(* IEC 61131-3 sources: PLC_structured_text/, 3 files *)

(* ---- electrical_motor.st ---- *)
PROGRAM Main
VAR
	AI_FRQ	AT %IW2: INT;
	AO_FRQ	AT %QW2: INT;
	DI_RUN	AT %IX0.0: BOOL;
	DI_ERR	AT %IX0.1: BOOL;
	DI_AUTO	AT %IX0.2: BOOL;
	DO_RUN	AT %QX0.0: BOOL;
	DO_FWD	AT %QX0.4: BOOL;
	DO_BKW	AT %QX0.5: BOOL;
	EN_AI_HZ	AT %QX1.1: BOOL;
	Control_Mode	AT %MW0: INT;
	HMI_SHOW_Hz	AT %MW1: INT;
	HMI_SHOW_Err	AT %MW2: INT;
	HMI_SHOW_RUN	AT %MW3: INT;
	HMI_SHOW_NONE	AT %MW4: INT;
	HMI_SET_FWD	AT %MW6: INT;
	HMI_SET_BCK	AT %MW7: INT;
	HMI_SET_Fr_GiveAQ AT %MW10: INT;
	RUN_TIME AT %MD11: REAL;
	HMI_SET_FR	AT %MD12: REAL;
	CurveSet_Hz	: REAL;
	CurveSet_Count : DINT;
	BLINK01 : BLINK;
	BLINK02 : BLINK;
	BLINK03 : BLINK;
	R_TRIG01 : R_TRIG;
	R_TRIG02 : R_TRIG;
	R_TRIG03 : R_TRIG;

	Run_count: DINT;
	Run_fre: REAL;
END_VAR

HMI_SHOW_Hz	:= AI_FRQ;
IF HMI_SET_FR >= 0.0 AND HMI_SET_FR <= 50.0 THEN
	HMI_SET_Fr_GiveAQ := REAL_TO_INT(HMI_SET_FR * 100.0);
END_IF
CASE control_mode OF
	1: AO_FRQ := HMI_SET_Fr_GiveAQ;
	2: AO_FRQ := REAL_TO_INT(Run_fre);
	3: AO_FRQ := REAL_TO_INT(CurveSet_Hz);
	4: AO_FRQ := REAL_TO_INT(Run_fre);
	0: AO_FRQ := 0;
END_CASE

EN_AI_HZ := (control_mode = 1) OR (control_mode = 3) OR (control_mode = 2) OR (control_mode = 4);

HMI_SHOW_Err := BOOL_TO_INT(DI_ERR);
HMI_SHOW_RUN := BOOL_TO_INT(DI_RUN);
HMI_SHOW_NONE := BOOL_TO_INT(DI_AUTO);
DO_RUN := INT_TO_BOOL(HMI_SET_FWD) OR INT_TO_BOOL(HMI_SET_BCK);
DO_FWD := INT_TO_BOOL(HMI_SET_FWD);
DO_BKW := INT_TO_BOOL(HMI_SET_BCK);

BLINK01(ENABLE := (control_mode = 3) , TIMELOW := T#50MS, TIMEHIGH:= T#50MS, OUT => );
BLINK02(ENABLE := (control_mode = 2) , TIMELOW := T#50MS, TIMEHIGH:= T#50MS, OUT => );
BLINK03(ENABLE := (control_mode = 4) , TIMELOW := T#50MS, TIMEHIGH:= T#50MS, OUT => );

R_TRIG01(CLK := BLINK01.OUT, Q => );
R_TRIG02(CLK := BLINK02.OUT, Q => );
R_TRIG03(CLK := BLINK03.OUT, Q => );

IF (control_mode = 0) THEN
	Run_fre := 0.0;
	RUN_TIME := 0.0;
	Run_count := 0;
	CurveSet_Count := 0;
END_IF

IF (control_mode = 2) THEN
	Run_fre := 4500.0;
	HMI_SET_FWD := BOOL_TO_INT(Run_count <= 600);
	HMI_SET_BCK := BOOL_TO_INT((Run_count > 600) AND (Run_count <= 1200));
	IF Run_count > 1200 THEN
		Run_fre := 0.0;
		Run_count := 0;
		RUN_TIME := 0.0;
		control_mode := 0;
	END_IF
END_IF

IF R_TRIG02.Q AND Run_Count <= 1200 THEN
	Run_count := Run_count + 1;
	RUN_TIME := RUN_TIME + 1;
END_IF

IF (control_mode = 3) THEN
	HMI_SET_FWD := BOOL_TO_INT((CurveSet_Count <= 1800) AND (CurveSet_Count >0));
END_IF

IF R_TRIG01.Q AND CurveSet_Count <= 1800 THEN
	IF (CurveSet_Count = 0) THEN
		CurveSet_Hz := 0.0;
	END_IF
	CurveSet_Count := CurveSet_Count + 1;
	RUN_TIME := RUN_TIME + 1;

	IF CurveSet_Count > 0 AND CurveSet_Count <= 450 THEN
		CurveSet_Hz := CurveSet_Hz + (2500.0/450.0);
	END_IF
	IF CurveSet_Count > 450 AND CurveSet_Count <= 600 THEN
		CurveSet_Hz := CurveSet_Hz - (2500.0/150.0);
	END_IF
	IF CurveSet_Count > 600 AND CurveSet_Count <= 900 THEN
		CurveSet_Hz := CurveSet_Hz + (2500.0/300.0);
	END_IF
	IF CurveSet_Count > 900 AND CurveSet_Count <= 1200 THEN
		CurveSet_Hz := CurveSet_Hz - (2500.0/300.0);
	END_IF
	IF CurveSet_Count > 1200 AND CurveSet_Count <= 1500 THEN
		CurveSet_Hz := CurveSet_Hz + (2500.0/300.0);
	END_IF
	IF CurveSet_Count > 1500 AND CurveSet_Count <= 1800 THEN
		CurveSet_Hz := CurveSet_Hz - (2500.0/300.0);
	END_IF
	IF CurveSet_Count > 1800 THEN
		CurveSet_Count := 0;
		CurveSet_Hz := 0.0;
		RUN_TIME := 0.0;
		control_mode := 0;
	END_IF
END_IF

IF R_TRIG03.Q THEN
	Run_count := Run_count + 1;
	RUN_TIME := RUN_TIME + 1;
END_IF

IF (control_mode = 4) THEN
	HMI_SET_FWD := 1;
	IF Run_count MOD 100 = 0 THEN
		IF Run_fre <= 4500 THEN
			//Run_fre := Run_fre + 16.6;
			Run_fre := Run_count;
		END_IF
	END_IF
END_IF

(* ---- electroplating_production_line.st ---- *)
PROGRAM Main
VAR
    left_strict AT %IX0.0: BOOL;
    first_place AT %IX0.1: BOOL;
    second_place AT %IX0.2: BOOL;
    third_place AT %IX0.3: BOOL;
    right_strict AT %IX0.4: BOOL;
    up_strict AT %IX0.5: BOOL;
    down_strict AT %IX0.6: BOOL;

    left AT %QX0.0: BOOL;
    right AT %QX0.1: BOOL;
    up AT %QX0.2: BOOL;
    down AT %QX0.3: BOOL;

    left_temp: BOOL;
    right_temp: BOOL;
    up_temp: BOOL;
    down_temp: BOOL;
    status_temp : INT;

    status AT %MW0: INT; //0 stop ; 1 auto;  2 manual; 3 reset; 4
    pause AT %MX30.0: BOOL;
    run_count AT %MW1: INT;
    run_count_set AT%MX4.0: BOOL;
    run_count_strict: INT;
    time_show AT %MW3: INT;

    HMI_left_strict AT %MX20.0: BOOL;
    HMI_mid_1 AT %MX21.0: BOOL; // MW1:X8
    HMI_first_place AT %MX20.1: BOOL;
    HMI_mid_2 AT %MX21.1: BOOL;
    HMI_second_place AT %MX20.2: BOOL;
    HMI_mid_3 AT %MX21.2: BOOL;
    HMI_third_place AT %MX20.3: BOOL;
    HMI_mid_4 AT %MX21.3: BOOL;
    HMI_right_strict AT %MX20.4: BOOL;

    HMI_up_strict AT %MX20.5: BOOL;
    HMI_down_strict AT %MX20.6: BOOL;

    HMI_RUN_status AT %MX22.1: BOOL;
    HMI_STOP_status AT %MX22.2: BOOL;
    HMI_RESET_status AT %MX22.3: BOOL;

    HMI_left AT%MX24.0: BOOL;
    HMI_right AT%MX24.1: BOOL;
    HMI_up AT%MX24.2: BOOL;
    HMI_down AT%MX24.3: BOOL;

    mid_1: BOOL;
    mid_2: BOOL;
    mid_3: BOOL;
    mid_4: BOOL;

    pass_left_strict: BOOL;
    pass_first_place: BOOL;
    pass_second_place: BOOL;
    pass_third_place: BOOL;
    pass_right_strict: BOOL;
    pass_up_strict: BOOL;
    pass_down_strict: BOOL;
    h_direction : INT; // 1 left; 2 right;
    v_direction : INT; // 1 up; 2 down;

    first_place_time: INT;
    first_place_stand_time: INT;
    second_place_time: INT;
    second_place_stand_time: INT;
    third_place_time: INT;
    third_place_stand_time: INT;

    current_basic_time: INT;
    start_timing: BOOL;
    temp_time: INT;

    right_progress: BOOL;
    down_to_strict : BOOL;
    up_to_strict : BOOL;
    already_down : BOOL;
    auto_mode_reset : BOOL;

    BLINK_1: BLINK;
    TRIG_1: R_TRIG;

END_VAR

BLINK_1(ENABLE := (status = 1 OR status = 2) , TIMELOW := T#500MS, TIMEHIGH:= T#500MS, OUT => );
TRIG_1(CLK := BLINK_1.OUT, Q => );

first_place_time := 10;
first_place_stand_time := 3;
second_place_time := 8;
second_place_stand_time := 3;
third_place_time := 5;
third_place_stand_time := 3;

IF pause THEN
    // store value
    left_temp := left;
    right_temp := right;
    up_temp := up;
    down_temp := down;
    status_temp := status;
    // set to sotp
    status := 4;
    left := FALSE;
    right := FALSE;
    up := FALSE;
    down := FALSE;
ELSIF (NOT pause) AND status = 4 THEN
    // restore value
    left := left_temp;
    right := right_temp;
    up := up_temp;
    down := down_temp;
    status := status_temp;
END_IF

// place control
IF left_strict THEN
    pass_left_strict := TRUE;
    pass_first_place := FALSE;
    pass_second_place := FALSE;
    pass_third_place := FALSE;
    pass_right_strict := FALSE;
    pass_up_strict := FALSE;
    pass_down_strict := FALSE;
END_IF
IF pass_left_strict THEN
    mid_1 := TRUE;
END_IF

IF status = 0 THEN
    HMI_RUN_status := FALSE;
    HMI_STOP_status := TRUE;
    HMI_RESET_status := FALSE;
    h_direction := 0;
    v_direction := 0;
    run_count := 0;
    time_show := 0;
    left := FALSE;
    right := FALSE;
    up := FALSE;
    down := FALSE;
END_IF

// when status = 1 or 2 mark start
IF status = 1 OR status = 2 THEN
    HMI_RUN_status := TRUE;
    HMI_STOP_status := FALSE;
    HMI_RESET_status := FALSE;
END_IF

IF status = 3 THEN
    HMI_RUN_status := FALSE;
    HMI_STOP_status := FALSE;
    HMI_RESET_status := TRUE;
END_IF

IF status = 3 THEN
    //run_count := 0;
    time_show := 0;
    IF left_strict = FALSE THEN
        left := TRUE;
        h_direction := 1;
    ELSE
        left := FALSE;
    END_IF
    IF up_strict = FALSE THEN
        up := TRUE;
        v_direction := 1;
    ELSE
        up := FALSE;
    END_IF
    IF left_strict AND up_strict THEN
        status := 0;
    END_IF
END_IF

IF status = 2 THEN
    IF NOT up_strict THEN
        IF HMI_up THEN
            up := TRUE;
            v_direction := 1;
        ELSE
            up := FALSE;
        END_IF
    END_IF
    IF NOT down_strict THEN
        IF HMI_down THEN
            down := TRUE;
            v_direction := 2;
        ELSE
            down := FALSE;
        END_IF
    END_IF
    IF NOT left_strict THEN
        IF HMI_left THEN
            left := TRUE;
            h_direction := 1;
        ELSE
            left := FALSE;
        END_IF
    END_IF
    IF NOT right_strict THEN
        IF HMI_right THEN
            right := TRUE;
            h_direction := 2;
        ELSE
            right := FALSE;
        END_IF
    END_IF
END_IF

IF run_count_set THEN
    run_count_strict := 1;
ELSIF NOT run_count_set THEN
    run_count_strict := -1;
END_IF

IF status = 1 THEN
    IF run_count = run_count_strict THEN
        status := 3;
    ELSE
        IF left_strict THEN
            auto_mode_reset := FALSE;
            left := FALSE;
            right_progress := TRUE;
        END_IF

        IF right_progress THEN
            right := TRUE;
            h_direction := 2;
        ELSIF NOT right_progress THEN
            right := FALSE;
        END_IF

        IF first_place THEN
            right_progress := FALSE;

            IF down_strict THEN
                start_timing := TRUE;
                current_basic_time := first_place_time;
                IF time_show = 0 THEN
                    start_timing := FALSE;
                    already_down := TRUE;
                END_IF
            ELSIF (NOT down_strict) AND (NOT already_down) THEN
                down := TRUE;
                v_direction := 2;
            END_IF

            IF already_down THEN
                IF up_strict THEN
                    start_timing := TRUE;
                    current_basic_time := first_place_stand_time;
                    IF time_show = 0 THEN
                        start_timing := FALSE;
                        already_down := FALSE;
                        right_progress := TRUE;
                    END_IF
                ELSE
                    up := TRUE;
                    v_direction := 1;
                END_IF
            END_IF
        END_IF

        IF second_place THEN
            right_progress := FALSE;

            IF down_strict THEN
                start_timing := TRUE;
                current_basic_time := second_place_time;
                IF time_show = 0 THEN
                    start_timing := FALSE;
                    already_down := TRUE;
                END_IF
            ELSIF (NOT down_strict) AND (NOT already_down) THEN
                down := TRUE;
                v_direction := 2;
            END_IF

            IF already_down THEN
                IF up_strict THEN
                    start_timing := TRUE;
                    current_basic_time := second_place_stand_time;
                    IF time_show = 0 THEN
                        start_timing := FALSE;
                        already_down := FALSE;
                        right_progress := TRUE;
                    END_IF
                ELSE
                    up := TRUE;
                    v_direction := 1;
                END_IF
            END_IF
        END_IF

        IF third_place THEN
            right_progress := FALSE;

            IF down_strict THEN
                start_timing := TRUE;
                current_basic_time := third_place_time;
                IF time_show = 0 THEN
                    start_timing := FALSE;
                    already_down := TRUE;
                END_IF
            ELSIF (NOT down_strict) AND (NOT already_down) THEN
                down := TRUE;
                v_direction := 2;
            END_IF

            IF already_down THEN
                IF up_strict THEN
                    start_timing := TRUE;
                    current_basic_time := third_place_stand_time;
                    IF time_show = 0 THEN
                        start_timing := FALSE;
                        already_down := FALSE;
                        right_progress := TRUE;
                    END_IF
                ELSE
                    up := TRUE;
                    v_direction := 1;
                END_IF
            END_IF
        END_IF

        IF right_strict THEN
            run_count := run_count + 1;
            right_progress := FALSE;
            auto_mode_reset := TRUE;
        END_IF

        IF auto_mode_reset THEN
            left := TRUE;
            h_direction := 1;
        END_IF
    END_IF
END_IF

IF TRIG_1.Q THEN
    IF start_timing AND (NOT pause) THEN
        temp_time := temp_time + 1;
        time_show := current_basic_time - temp_time;
    ELSIF NOT start_timing THEN
        time_show := 0;
        temp_time := 0;
    END_IF
END_IF

(* ---- traffic_light_control.st ---- *)
PROGRAM Main
VAR
    first_button_g AT %IX0.0: BOOL;  // start
    first_button_y AT %IX0.1: BOOL;
    first_button_r AT %IX0.2: BOOL; //  stop
    second_button_g AT %IX0.3: BOOL;
    second_button_y AT %IX0.4: BOOL;
    second_button_r AT %IX0.5: BOOL;

    ns_car_r AT %QX0.0: BOOL;
    ns_car_y AT %QX0.1: BOOL;
    ns_car_g AT %QX0.2: BOOL;

    we_car_r AT %QX0.3: BOOL;
    we_car_y AT %QX0.4: BOOL;
    we_car_g AT %QX0.5: BOOL;

    ns_human_r AT %QX0.6: BOOL;
    ns_human_g AT %QX0.7: BOOL;

    we_human_r AT %QX0.8: BOOL;
    we_human_g AT %QX0.9: BOOL;

    HMI_ns_car_time AT %MW1: INT;
    HMI_we_car_time AT %MW2: INT;
    HMI_ns_human_time AT %MW3: INT;
    HMI_we_human_time AT %MW4: INT;

    HMI_ns_car_r AT %MX15.0: BOOL;
    HMI_ns_car_y AT %MX15.1: BOOL;
    HMI_ns_car_g AT %MX15.2: BOOL;
    HMI_ns_human_r AT %MX15.3: BOOL;
    HMI_ns_human_g AT %MX15.4: BOOL;

    HMI_we_car_r AT %MX16.0: BOOL;
    HMI_we_car_y AT %MX16.1: BOOL;
    HMI_we_car_g AT %MX16.2: BOOL;
    HMI_we_human_r AT %MX16.3: BOOL;
    HMI_we_human_g AT %MX16.4: BOOL;

    HMI_first_button_g AT %MX17.0: BOOL;
    HMI_first_button_y AT %MX17.1: BOOL;
    HMI_first_button_r AT %MX17.2: BOOL;
    HMI_second_button_g AT %MX18.0: BOOL;
    HMI_second_button_y AT %MX18.1: BOOL;
    HMI_second_button_r AT %MX18.2: BOOL;

    HMI_car_red_time AT %MW19: INT;
    HMI_car_green_time AT %MW20: INT;
    HMI_car_yellow_time AT %MW21: INT;
    HMI_TIME_SET AT %MX14.0: BOOL;

    ns_r_temp_time: INT;
    we_r_temp_time: INT;
    ns_g_temp_time: INT;
    we_g_temp_time: INT;
    ns_y_temp_time: INT;
    we_y_temp_time: INT;
    ns_human_temp_time: INT;
    we_human_temp_time: INT;
    start: BOOL;
    stop: BOOL;

    car_red_time: INT;
    car_yellow_time: INT;
    car_green_time: INT;
    human_red_time: INT;
    human_green_time: INT;

    ns_car_go: BOOL;
    ns_car_stop: BOOL;
    ns_human_go: BOOL;
    ns_red: BOOL;
    ns_green: BOOL;
    ns_yellow: BOOL;

    we_car_go: BOOL;
    we_car_stop: BOOL;
    we_human_go: BOOL;
    we_red: BOOL;
    we_green: BOOL;
    we_yellow: BOOL;

    passer_button: BOOL;

    BLINK_1: BLINK;
    TRIG_1: R_TRIG;

END_VAR

// allow HMI set time
IF HMI_TIME_SET THEN
    car_red_time := HMI_car_red_time - 1;
    car_green_time := HMI_car_green_time - 1;
    car_yellow_time := HMI_car_red_time - HMI_car_green_time - 1;
    HMI_car_yellow_time := car_yellow_time + 1;
ELSE
    car_red_time := 19;
    car_green_time := 14;
    car_yellow_time := 4;
    HMI_car_red_time := car_red_time + 1;
    HMI_car_green_time := car_green_time + 1;
    HMI_car_yellow_time := car_yellow_time + 1;
END_IF

human_red_time := car_red_time + car_yellow_time + 1; //double 0 have been added, so
human_green_time := car_green_time;

// button triger
IF first_button_g THEN
    IF NOT start THEN
        ns_red := TRUE;
        we_green := TRUE;
        HMI_ns_human_time := car_red_time;
        HMI_we_human_time := human_green_time;
    END_IF
    start := TRUE;
    stop := FALSE;
END_IF

IF first_button_r THEN
    start := FALSE;
    stop := TRUE;
END_IF

IF second_button_g OR second_button_r THEN
    IF (ns_red AND we_green) OR (we_red AND ns_green) THEN
        passer_button := TRUE;
    END_IF
END_IF

// time relative
BLINK_1(ENABLE := (start = TRUE) , TIMELOW := T#500MS, TIMEHIGH:= T#500MS, OUT => );
TRIG_1(CLK := BLINK_1.OUT, Q => );

//bind
HMI_ns_car_r := ns_car_r;
HMI_ns_car_y := ns_car_y;
HMI_ns_car_g := ns_car_g;
HMI_ns_human_r := ns_human_r;
HMI_ns_human_g := ns_human_g;
HMI_we_car_r := we_car_r;
HMI_we_car_y := we_car_y;
HMI_we_car_g := we_car_g;
HMI_we_human_r := we_human_r;
HMI_we_human_g := we_human_g;
HMI_first_button_g := first_button_g;
HMI_first_button_y := first_button_y;
HMI_first_button_r := first_button_r;
HMI_second_button_g := second_button_g;
HMI_second_button_y := second_button_y;
HMI_second_button_r := second_button_r;

// clear
IF stop THEN
    ns_r_temp_time := 0;
    we_r_temp_time := 0;
    ns_g_temp_time := 0;
    we_g_temp_time := 0;
    we_y_temp_time := 0;
	ns_y_temp_time := 0;
    ns_human_temp_time := 0;
    we_human_temp_time := 0;
    we_red := FALSE;
    we_green := FALSE;
    we_yellow := FALSE;
    ns_red := FALSE;
    ns_green := FALSE;
    ns_yellow := FALSE;
    ns_car_go := FALSE;
    we_car_go := FALSE;
    ns_human_go := FALSE;
    we_human_go := FALSE;
    we_car_r := FALSE;
    we_car_y := FALSE;
    we_car_g := FALSE;
    we_human_g := FALSE;
    we_human_r := FALSE;
    ns_car_r := FALSE;
    ns_car_y := FALSE;
    ns_car_g := FALSE;
    ns_human_g := FALSE;
    ns_human_r := FALSE;
    HMI_ns_car_time := 0;
    HMI_ns_human_time := 0;
    HMI_we_car_time := 0;
    HMI_we_human_time := 0;
END_IF

// time

IF ns_red THEN
    ns_car_go := FALSE;
    ns_human_go := FALSE;
    IF ns_r_temp_time = car_red_time + 1 THEN // 19 equals to 20 second because of 0
        ns_r_temp_time := 0;
        HMI_ns_car_time := car_green_time;

        ns_human_temp_time := 0;
        HMI_ns_human_time := human_green_time;

        ns_red := FALSE;
        ns_green := TRUE;
    END_IF
END_IF

IF we_red THEN
    we_car_go := FALSE;
    we_human_go := FALSE;
    IF we_r_temp_time = car_red_time + 1 THEN
        we_r_temp_time := 0;
        HMI_we_car_time := car_green_time;

        we_human_temp_time := 0;
        HMI_we_human_time := human_green_time;

        we_red:= FALSE;
        we_green := TRUE;
    END_IF
END_IF

IF ns_car_go THEN
    ns_car_r := FALSE;
    ns_car_g := TRUE;
ELSIF (NOT ns_car_go AND start) THEN
    ns_car_r := TRUE;
    ns_car_g := FALSE;
END_IF

IF we_car_go THEN
    we_car_r := FALSE;
    we_car_g := TRUE;
ELSIF (NOT we_car_go AND start) THEN
    we_car_r := TRUE;
    we_car_g := FALSE;
END_IF

IF ns_human_go THEN
    ns_human_g := TRUE;
    ns_human_r := FALSE;
ELSIF (ns_human_go = FALSE AND start = TRUE) THEN
    ns_human_g := FALSE;
    ns_human_r := TRUE;
END_IF;

IF we_human_go THEN
    we_human_g := TRUE;
    we_human_r := FALSE;
ELSIF (we_human_go = FALSE AND start = TRUE) THEN
    we_human_g := FALSE;
    we_human_r := TRUE;
END_IF;

IF ns_green THEN
    ns_car_go := TRUE;
    ns_human_go := TRUE;
    IF car_green_time + 1 - ns_g_temp_time <= 4 THEN
        IF ns_g_temp_time MOD 2 = 1 THEN
            ns_car_g := FALSE;
        END_IF
    END_IF
    IF ns_g_temp_time = car_green_time + 1 THEN
        ns_g_temp_time := 0;
        HMI_ns_car_time := car_yellow_time;

        ns_human_temp_time := 0;
        HMI_ns_human_time := human_red_time;

        ns_yellow := TRUE;
        ns_green := FALSE;
    END_IF
END_IF

IF we_green THEN
    we_car_go := TRUE;
    we_human_go := TRUE;
    IF car_green_time + 1 - we_g_temp_time <= 4 THEN
        IF we_g_temp_time MOD 2 = 1 THEN
            we_car_g := FALSE;
        END_IF
    END_IF
    IF we_g_temp_time = car_green_time + 1 THEN
        we_g_temp_time := 0;
        HMI_we_car_time := car_yellow_time;

        we_human_temp_time := 0;
        HMI_we_human_time := human_red_time;

        we_yellow := TRUE;
        we_green := FALSE;
    END_IF
END_IF

IF ns_yellow THEN
    ns_car_y := TRUE;
    ns_car_g := FALSE;
    ns_car_r := FALSE;
    ns_human_go := FALSE;
    IF ns_y_temp_time = car_yellow_time + 1 THEN
        ns_y_temp_time := 0;
        HMI_ns_car_time := car_red_time;

        ns_car_y := FALSE;
        ns_yellow := FALSE;
        ns_red := TRUE;
    END_IF
    //
END_IF

IF we_yellow THEN
    we_car_y := TRUE;
    we_car_r := FALSE;
    we_car_g := FALSE;
    we_human_go := FALSE;
    IF we_y_temp_time = car_yellow_time + 1 THEN
        we_y_temp_time := 0;
        HMI_we_car_time := car_red_time;

        we_car_y := FALSE;
        we_yellow := FALSE;
        we_red := TRUE;
	END_IF
END_IF

// passer_button
IF passer_button THEN
    IF ns_red AND we_green AND ns_r_temp_time + 3 <= car_red_time + 1 AND we_g_temp_time + 3 <= car_green_time + 1 THEN
        ns_r_temp_time := ns_r_temp_time + 3;
        we_g_temp_time := we_g_temp_time + 3;
        ns_human_temp_time := ns_human_temp_time + 3;
        we_human_temp_time := we_human_temp_time + 3;
    END_IF
    IF we_red AND ns_green AND we_r_temp_time + 3 <= car_red_time + 1 AND ns_g_temp_time + 3 <= car_green_time + 1 THEN
        we_r_temp_time := we_r_temp_time + 3;
        ns_g_temp_time := ns_g_temp_time + 3;
        ns_human_temp_time := ns_human_temp_time + 3;
        we_human_temp_time := we_human_temp_time + 3;
    END_IF
    passer_button := FALSE;
END_IF

IF TRIG_1.Q THEN
    IF ns_red THEN
        ns_r_temp_time := ns_r_temp_time + 1;
        HMI_ns_car_time := car_red_time - ns_r_temp_time;
    END_IF
    IF we_red THEN
        we_r_temp_time := we_r_temp_time + 1;
        HMI_we_car_time := car_red_time - we_r_temp_time;
    END_IF
    IF ns_green THEN
        ns_g_temp_time := ns_g_temp_time + 1;
        HMI_ns_car_time := car_green_time - ns_g_temp_time;
    END_IF
    IF we_green THEN
        we_g_temp_time := we_g_temp_time + 1;
        HMI_we_car_time := car_green_time - we_g_temp_time;
    END_IF
    IF ns_yellow THEN
        ns_y_temp_time := ns_y_temp_time + 1;
        HMI_ns_car_time := car_yellow_time - ns_y_temp_time;
    END_IF
    IF we_yellow THEN
        we_y_temp_time := we_y_temp_time + 1;
        HMI_we_car_time := car_yellow_time - we_y_temp_time;
    END_IF
    // human
    IF (ns_human_go AND ns_green) THEN
        ns_human_temp_time := ns_human_temp_time + 1;
        HMI_ns_human_time := human_green_time - ns_human_temp_time;
    END_IF
    IF (NOT ns_human_go AND NOT ns_green)THEN
        ns_human_temp_time := ns_human_temp_time + 1;
        HMI_ns_human_time := human_red_time - ns_human_temp_time;
    END_IF
    IF (we_human_go AND we_green) THEN
        we_human_temp_time := we_human_temp_time + 1;
        HMI_we_human_time := human_green_time - we_human_temp_time;
    END_IF
    IF (NOT we_human_go AND NOT we_green) THEN
        we_human_temp_time := we_human_temp_time + 1;
        HMI_we_human_time := human_red_time - we_human_temp_time;
    END_IF
END_IF
